FUNCTION_BLOCK JSON_PARSER_2442D0DD1B0E13218 (* Generic Interface Function Block Type *)
  (* Standard: 61499-2 *)
  (* Version 0.0, 30/03/2021, SESA471728, Schneider Electric, Template *)
  PACKAGE UAO.Hackathon;
  (* Compiler Cpp nxtControl builtin 1.0 *)
  {SET_ATTRIBUTE(Runtime.FBType.ImplementingType, Runtime.Standard#DYNGEN_JSON_PARSER)}
  {SET_ATTRIBUTE(Configuration.GenericFBType.InterfaceParams, Runtime.Base#CNT:=2;valueOut${CNT$}:STRING,STRING)}
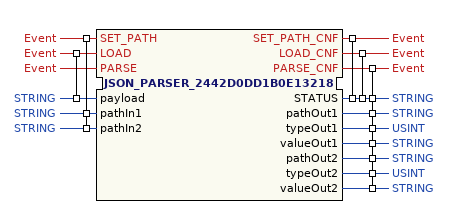
  EVENT_INPUT
    SET_PATH WITH pathIn1, pathIn2; (* Event dedicated for JSON path management *)
    LOAD WITH payload; (* Event dedicated for payload management *)
    PARSE; (* Event dedicated for parse payload management *)
  END_EVENT
  EVENT_OUTPUT
    SET_PATH_CNF WITH STATUS; (* Confirmation for JSON path management event *)
    LOAD_CNF WITH STATUS; (* Confirmation for payload management event *)
    PARSE_CNF WITH STATUS, pathOut1, pathOut2, typeOut1, typeOut2, valueOut1, valueOut2; (* Confirmation for json parse management event *)
  END_EVENT
  VAR_INPUT
    payload : STRING; (* JSON payload to parse *)
    pathIn1 : STRING; (* JSON path *)
    pathIn2 : STRING; (* JSON path *)
  END_VAR
  VAR_OUTPUT
    STATUS : STRING; (* Status *)
    pathOut1 : STRING; (* JSON output path *)
    typeOut1 : USINT; (* Type of the output value *)
    valueOut1 : STRING; (* Output value *)
    pathOut2 : STRING; (* JSON output path *)
    typeOut2 : USINT; (* Type of the output value *)
    valueOut2 : STRING; (* Output value *)
  END_VAR
  EC_STATES
    START;
  END_STATES
END_FUNCTION_BLOCK
